Staubli VAL3: debug.pgx

public program debug(num& x_nExecStatus)
begin

  // Do nothing - not needed on CS9

end
